INTERFACE I_Flag EXTENDS Debug.I_Debug, Tags.I_Tagged

METHOD IsLowered : BOOL
VAR_INPUT
END_VAR
END_METHOD

METHOD IsRised : BOOL
VAR_INPUT
END_VAR
END_METHOD

PROPERTY Tag : Tags.I_Tag
GET
END_GET
END_PROPERTY

END_INTERFACE

(* stored: Version 1.1.0.1
   Itf I_Flag: Id {8923833a-63ee-4bdd-8989-492b2c0dec51}
   Method IsLowered: Id {80fd9e90-471e-4626-8311-270df904b500}
   Method IsRised: Id {f5d2728d-de30-45bf-99f3-6800a8dbc690}
   Property Tag: Id {105135e3-c17a-46a0-825e-a8b7bf61063e}
   Get Get: Id {e2c1591c-f789-472e-ba5a-c393968e67f1} *)
